{attribute 'no_explicit_call' := 'do not call this POU directly'} 
FUNCTION_BLOCK DigitalInput IMPLEMENTS I_DigitalChannel
VAR_INPUT
END_VAR
VAR_OUTPUT
END_VAR
VAR
    {attribute 'TcInitSymbol'}
	ID:				STRING(25);
	Channel			AT%I*: BOOL;
END_VAR

PROPERTY PUBLIC P_ID : String(25)
GET
P_ID:= ID;
END_GET
END_PROPERTY

PROPERTY P_State : EPlcMappingStatus
GET
P_State:= F_GetMappingStatus(adr(Channel), sizeof(BOOL));
END_GET
END_PROPERTY

PROPERTY PUBLIC P_Value : bool
GET
P_Value:= Channel;
END_GET
SET // PUBLIC
Channel:= P_Value;
END_SET
END_PROPERTY

END_FUNCTION_BLOCK

(* stored: Version 1.1.0.1
   POU DigitalInput: Id {8904ca26-c33a-0d5e-01bd-927c832f4cd0}, SpecialFunc None
   Property P_ID: Id {d2592e33-0c09-00ed-2a19-2a2ac1387854}
   Get Get: Id {db03f916-1db4-0ef0-2610-a102e9e38d81}
   Property P_State: Id {c3d8c2a3-d582-03a1-3305-487cd866c231}
   Get Get: Id {d84261ad-8c83-064f-0dc4-445397d3c6cc}
   Property P_Value: Id {eb10c2b4-f572-0e2d-2bec-edb3aca0020c}
   Get Get: Id {0af5f71f-a62f-0bc9-1f1b-442ea0defb72}
   Set Set: Id {a5ae33fe-bcc6-09a5-0371-0da6975e192e} *)
